(* IEC 61131-3 sources: programs/VI-54/VI-54_20171205/VI-54_20171205/Stations/Screen/LseClass170718/Class/SendDataCMD_PLC, 1 file *)

(* ---- SendDataCMD_PLC.st ---- *)
(*!
<Class
	Name               = "SendDataCMD_PLC"
	Revision           = "1.0"
	RealtimeTask       = "false"
	CyclicTask         = "true"
	BackgroundTask     = "true"
	Sigmatek           = "false"
	OSInterface        = "false"
	HighPriority       = "false"
	Automatic          = "false"
	UpdateMode         = "Prescan"
	SharedCommandTable = "true"
	Objectsize         = "(486,120)"
	Comment            = "Class passes the JobState and the JobID to the DiagnosticWork_PLC class.">
	<Channels>
		<Client Name="cStation" Required="true" Internal="false" Comment="Object channel to DiagnosticWork_PLC."/>
	</Channels>
	<RevDoku>
		<Owner Company="Sigmatek"/>
		<Dokumentation Revision="1.0" Date="2016-06-02" Author="HötAnt" Company="Sigmatek" Description="Creation"/>
	</RevDoku>
	<Network Name="SendDataCMD_PLC">
		<!-- List of Components in this network -->
		<Components>
			<Object
				Name       = "_base"
				Class      = "TCPComSend"
				Position   = "(218,120)"
				Visualized = "false">
				<Channels>
					<Server Name="ClassSvr"/>
					<Server Name="ID_Destination"/>
					<Server Name="ID_Source"/>
					<Server Name="sSendCnt"/>
					<Server Name="sSendErr"/>
					<Client Name="cPrio"/>
					<Client Name="cSendErr"/>
					<Client Name="cSendOk"/>
					<Client Name="toDataManager"/>
				</Channels>
			</Object>
		</Components>
		<Comments>
		</Comments>
		<!-- List of Connections in this network -->
		<Connections>
			<Connection Source="this.ClassSvr" Destination="_base.ClassSvr" Vertices="(1006,210),(834,210),"/>
			<Connection Source="this.ID_Destination" Destination="_base.ID_Destination" Vertices="(1006,270),(834,270),"/>
			<Connection Source="this.ID_Source" Destination="_base.ID_Source" Vertices="(1006,330),(834,330),"/>
			<Connection Source="this.sSendCnt" Destination="_base.sSendCnt" Vertices="(1006,390),(834,390),"/>
			<Connection Source="this.sSendErr" Destination="_base.sSendErr" Vertices="(1006,450),(834,450),"/>
			<Connection Source="_base.toDataManager" Destination="this.toDataManager" Vertices="(218,210),(38,210),"/>
			<Connection Source="_base.cPrio" Destination="this.cPrio" Vertices="(218,270),(38,270),"/>
		</Connections>
		<!-- Headerfiles -->
		<Options>
		</Options>
	</Network>
</Class>
*)
#pragma using TCPComSend

SendDataCMD_PLC : CLASS
: TCPComSend
  //Servers:
  //Clients:
	cStation 	: CltChCmd_DiagnosticWork_PLC;
  //Variables:
  //Functions:
				//! <Function Comment="Is called everytime the state of a job is changing. Overwrite to react to state changes." Name="CallBackJobState"/>
	FUNCTION VIRTUAL GLOBAL CallBackJobState
		VAR_INPUT
			JobID 	: DINT;
			JobState 	: DataManagerPriority::t_e_CallbackState;
		END_VAR;
  //Tables:
	FUNCTION @STD
		VAR_OUTPUT
			ret_code	: CONFSTATES;
		END_VAR;
	FUNCTION GLOBAL TAB @CT_;
END_CLASS;

#pragma usingLtd DiagnosticWork_PLC

// Ableitung ist notwendig , um den JobState an die Classe weiterzugeben.

FUNCTION VIRTUAL GLOBAL SendDataCMD_PLC::CallBackJobState
	VAR_INPUT
		JobID 	: DINT;
		JobState 	: DataManagerPriority::t_e_CallbackState;
	END_VAR

  // Base aufrufen , damit die Standard Server und Clients wie gewohnt aktualisiert werden.
  TCPComSend::CallBackJobState(JobID, JobState);

  case JobState of
    //Ok
    _MNG_Received:
       cStation.ResponseJobState(jobid,TRUE);

    //Error
    _MNG_NoReceiverConnected,
    _MNG_GlobalReceiveError,
    _MNG_TimeOut:
       cStation.ResponseJobState(jobid,FALSE);

  end_case;

END_FUNCTION
